GLOBALCONSTANTS colours (* Global constants *)
  (* Standard: 61499-1; Description: Copyright (c) 2023 HR Agrartechnik GmbH This program and the accompanying materials are made available under the terms of the Eclipse Public License 2.0 which is available at https://www.eclipse.org/legal/epl-2.0/ SPDX-License-Identifier: EPL-2.0 *)
  (* Version 1.0, 2023-10-22, Franz Höpfinger, HR Agrartechnik GmbH *)
  VAR_GLOBAL CONSTANT
    COLOR_BLACK : USINT := USINT#0;
    COLOR_WHITE : USINT := USINT#1;
    COLOR_GREEN : USINT := USINT#2;
    COLOR_TEAL : USINT := USINT#3;
    COLOR_MAROON : USINT := USINT#4;
    COLOR_PURPLE : USINT := USINT#5;
    COLOR_OLIVE : USINT := USINT#6;
    COLOR_SILVER : USINT := USINT#7;
    COLOR_GREY : USINT := USINT#8;
    COLOR_BLUE : USINT := USINT#9;
    COLOR_LIME : USINT := USINT#10;
    COLOR_CYAN : USINT := USINT#11;
    COLOR_RED : USINT := USINT#12;
    COLOR_MAGENTA : USINT := USINT#13;
    COLOR_YELLOW : USINT := USINT#14;
    COLOR_NAVY : USINT := USINT#15;
  END_VAR
END_GLOBALCONSTANTS
